FUNCTION Convert_DATE_TO_UINT : Hresult
VAR_INPUT
	in : DATE;
	out : REFERENCE TO UINT;
END_VAR
VAR
	converted : UINT;
END_VAR

converted := DATE_TO_UINT(in);

IF (UINT_TO_DATE(converted) <> in) THEN
	Convert_DATE_TO_UINT := INCOMPATIBLE;
	RETURN;
END_IF

out := converted;

END_FUNCTION

(* stored: Version 1.1.0.1, ProductVersion 3.1.4024.12
   POU Convert_DATE_TO_UINT: Id {43c367b2-bba1-41b5-bb76-9504feeee57e}, SpecialFunc None *)
